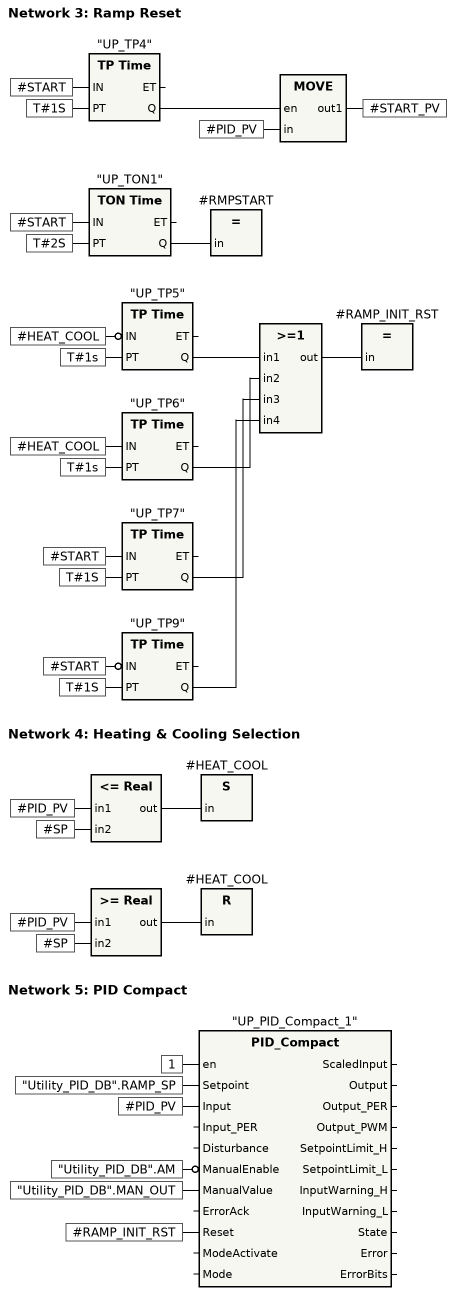
   "UP_TP4".TP(IN := #START, PT := T#1S);
   IF "UP_TP4".Q THEN #START_PV := #PID_PV; END_IF;
   "UP_TON1".TON(IN := #START, PT := T#2S);
   #RMPSTART := "UP_TON1".Q;
   "UP_TP5".TP(IN := NOT #HEAT_COOL, PT := T#1s);
   "UP_TP6".TP(IN := #HEAT_COOL, PT := T#1s);
   "UP_TP7".TP(IN := #START, PT := T#1S);
   "UP_TP9".TP(IN := NOT #START, PT := T#1S);
   #RAMP_INIT_RST := "UP_TP5".Q OR "UP_TP6".Q OR "UP_TP7".Q OR "UP_TP9".Q;
END_REGION

REGION Network 4: Heating & Cooling Selection
   // Heating & Cooling Selection
   IF #PID_PV <= #SP THEN #HEAT_COOL := TRUE; END_IF;
   IF #PID_PV >= #SP THEN #HEAT_COOL := FALSE; END_IF;
END_REGION

REGION Network 5: PID Compact
   IF 1 THEN
       "UP_PID_Compact_1"(Setpoint := "Utility_PID_DB".RAMP_SP,   // PID_Compact
                          Input := #PID_PV,
                          ManualEnable := NOT "Utility_PID_DB".AM,
                          ManualValue := "Utility_PID_DB".MAN_OUT,
                          Reset := #RAMP_INIT_RST);
   END_IF;
END_REGION

REGION Network 6 (SCL): Moving
   (* PID Parameters Moving *)
   "UP_PID_Compact_1".Retain.CtrlParams.Gain:= #P;
   "UP_PID_Compact_1".Retain.CtrlParams.Ti := #I;
   "UP_PID_Compact_1".Retain.CtrlParams.Td := #D;

   #RAMP := #SP;

   IF #RAMP_MODE OR #MASS_CONTROL THEN
       #PID_PV := #PV;
   END_IF;
   IF #JKT_RAMP THEN
       #PID_PV := #JAC_IN;
   END_IF;


   IF #AM = 1 AND #START = 1 AND #SOURCE_SEL<>5 THEN
       #SCVOUT := "UP_PID_Compact_1".Output;
       #CVOUT := "UP_PID_Compact_1".Output_PER;
   END_IF;
   IF (#AM = 1 AND #START = 0 ) OR (#AM = 1 AND #SOURCE_SEL=5) OR (#AM = 1 AND #START=1 AND (#AIR_XV_OPN OR #VENT_OPN OR #DRAIN_XV_OPN)) THEN
       #SCVOUT := 0.0;
       #CVOUT := 0;
   END_IF;
   IF #AM = 0 THEN
       #SCVOUT := "UP_PID_Compact_1".Output;
       #CVOUT := "UP_PID_Compact_1".Output_PER;
   END_IF;

   IF #AM = 1 AND #START = 1 AND #DRAIN_XV_OPN AND #SCV_XV_OPN THEN
       #iSTEAM_SCVOUT := 100.0;
       #iDRAIN_UP := 1;
   ELSE
       #iDRAIN_UP := 0;
   END_IF;
   IF #AM = 1 AND #START = 1 AND #SOURCE_SEL = 5 AND #iDRAIN_UP= 0 THEN
       #iSTEAM_SCVOUT := "UP_PID_Compact_1".Output;
       #iSTEAM_CVOUT := "UP_PID_Compact_1".Output_PER;
   END_IF;
   IF (#AM = 1 AND #START = 0) OR (#AM = 1 AND #SOURCE_SEL <> 5) OR (#AM = 1 AND #START = 1 AND ((#CONDENSATE_XV_OPN AND #SOURCE_SEL <> 5) OR (#AIR_XV_OPN AND #SOURCE_SEL = 5))) THEN
       #iSTEAM_SCVOUT := 0.0;
       #iSTEAM_CVOUT := 0;
   END_IF;


   (* Cooling *)
   IF #HEAT_COOL = 0 AND #START = 1 AND (#RAMP_MODE OR #JKT_RAMP) THEN
       "UP_RampFunction_DB1".PositiveFallingSlewRate := ABS((#START_PV - #SP) / (#TIME*60)); 
       "UP_PID_Compact_1".Config.InvertControl := 1;
   END_IF;
   IF #HEAT_COOL = 0 AND #START = 1 AND #MASS_CONTROL THEN
       "UP_RampFunction_DB1".PositiveFallingSlewRate := ABS((#START_PV - #SP) / (1 * 60));
       "UP_PID_Compact_1".Config.InvertControl := 1;
   END_IF;

   (* Heating *)
   IF #HEAT_COOL = 1 AND #START = 1 AND (#RAMP_MODE OR #JKT_RAMP) THEN
       "UP_RampFunction_DB1".PositiveRisingSlewRate := ABS((#SP - #START_PV) / (#TIME*60)); 
       "UP_PID_Compact_1".Config.InvertControl := 0;
   END_IF;
   IF #HEAT_COOL = 1 AND #START = 1 AND #MASS_CONTROL THEN
       "UP_RampFunction_DB1".PositiveRisingSlewRate := ABS((#SP - #START_PV) / (1 * 60));
       "UP_PID_Compact_1".Config.InvertControl := 0;
   END_IF;
END_REGION

REGION Network 7: OPERATION RUNTIME
   // OPERATION RUNTIME
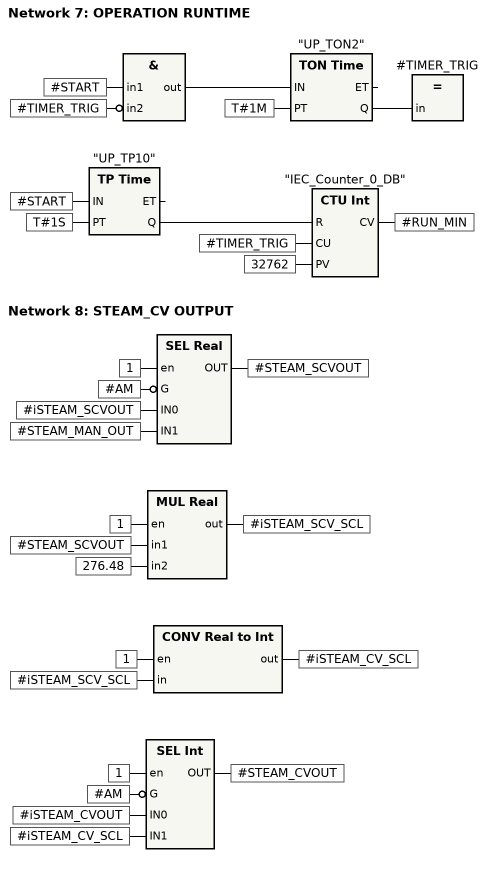
   "UP_TON2".TON(IN := #START AND NOT #TIMER_TRIG, PT := T#1M);
   #TIMER_TRIG := "UP_TON2".Q;
   "UP_TP10".TP(IN := #START, PT := T#1S);
   "IEC_Counter_0_DB".CTU(R := "UP_TP10".Q, CU := #TIMER_TRIG, PV := 32762, CV => #RUN_MIN);
END_REGION

REGION Network 8: STEAM_CV OUTPUT
   IF 1 THEN
       #STEAM_SCVOUT := SEL(G := NOT #AM, IN0 := #iSTEAM_SCVOUT, IN1 := #STEAM_MAN_OUT);
       #iSTEAM_SCV_SCL := #STEAM_SCVOUT * 276.48;
       #iSTEAM_CV_SCL := REAL_TO_INT(#iSTEAM_SCV_SCL);
       #STEAM_CVOUT := SEL(G := NOT #AM, IN0 := #iSTEAM_CVOUT, IN1 := #iSTEAM_CV_SCL);
   END_IF;
END_REGION
END_FUNCTION_BLOCK

FUNCTION_BLOCK "3WayValve"   // FB14, LAD
{ S7_Optimized_Access := 'TRUE' }
VERSION : 0.1
// stored: AutoNumber true, IsIECCheckEnabled false, IsRetainMemResEnabled false, MemoryReserve 100, SetENOAutomatically false, UDAEnableTagReadback false
   VAR_INPUT
      "auto/manual" : Bool;
      v1_open_auto : Bool;
      v1_open_man : Bool;
      v1_fbk_open : Bool;
      v1_fbk_close : Bool;
      v2_open_auto : Bool;
      v2_open_man : Bool;
      v2_fbk_open : Bool;
      reset : Bool;
      intl : Bool;
      monito_time : Time;
      Mon_En : Bool;
   END_VAR
   VAR_OUTPUT
      v1_cmd1 : Bool;
      v2_cmd2 : Bool;
      fault : Bool;
      status : Int;
   END_VAR
   VAR
      open_fault : Bool;
      close_fault : Bool;
      IEC_Timer_0_Instance : TON_TIME;
      IEC_Timer_0_Instance_1 { S7_SetPoint := 'True'} : TON_TIME;
      IEC_Timer_0_Instance_2 { S7_SetPoint := 'True'} : TON_TIME;
      V1_ON : Bool;
   END_VAR
   VAR_TEMP   // added for the SCL form of the ladder/FBD networks
      _w1 : Bool;
   END_VAR
BEGIN

REGION Network 1
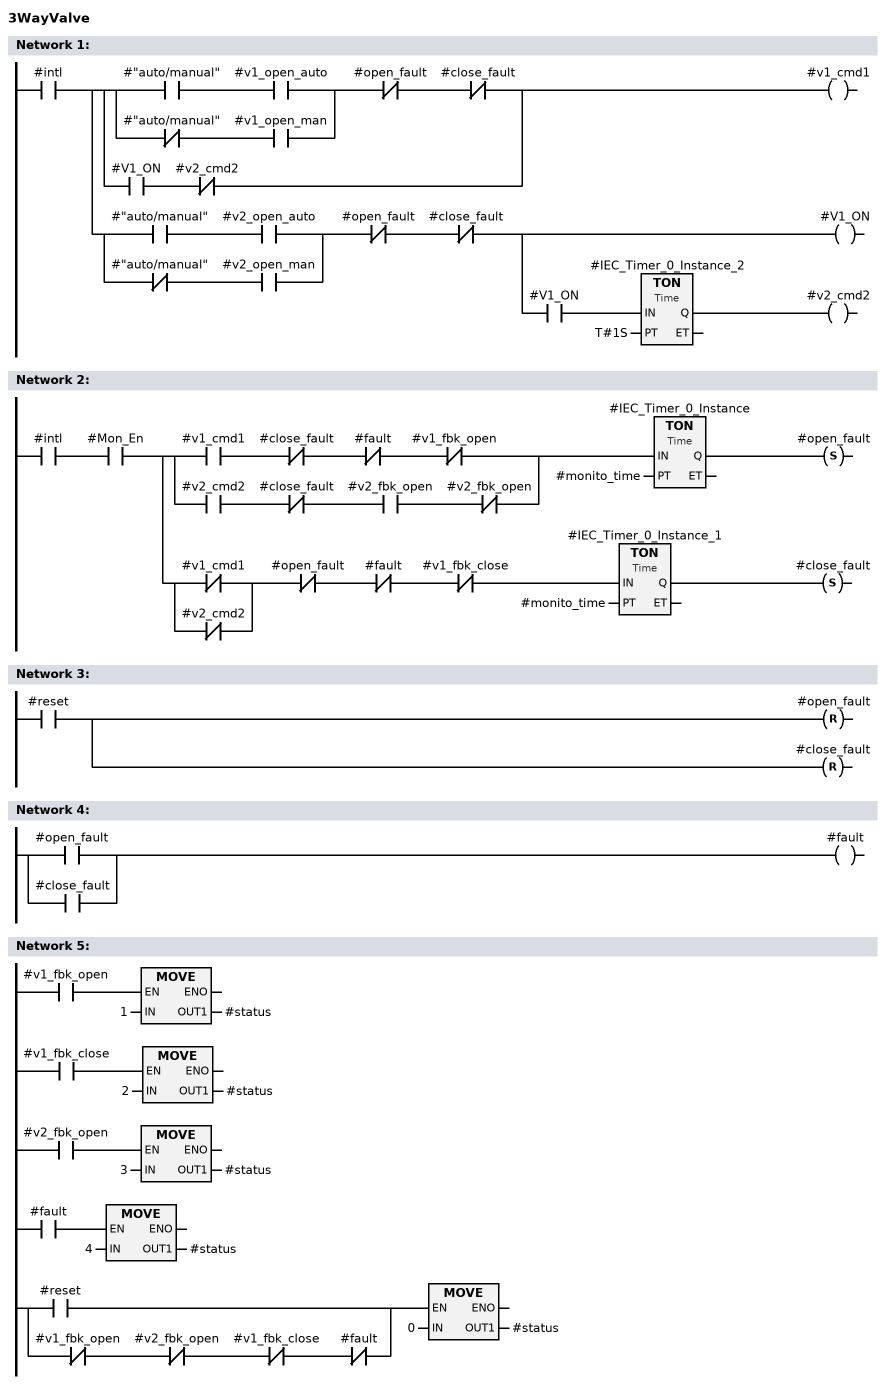
   RUNG wire#powerrail
      Contact( #intl )
      wire#w1
      Contact( #"auto/manual" )
      Contact( #v1_open_auto )
      wire#w2
      I_Contact( #open_fault )
      I_Contact( #close_fault )
      wire#w3
      Coil( #v1_cmd1 )
   END_RUNG
   RUNG wire#w1
      I_Contact( #"auto/manual" )
      Contact( #v1_open_man )
   END_RUNG wire#w2
   RUNG wire#w1
      Contact( #V1_ON )
      I_Contact( #v2_cmd2 )
   END_RUNG wire#w3
   RUNG wire#w1
      Contact( #"auto/manual" )
      Contact( #v2_open_auto )
      wire#w4
      I_Contact( #open_fault )
      I_Contact( #close_fault )
      wire#w5
      Coil( #V1_ON )
   END_RUNG
   RUNG wire#w1
      I_Contact( #"auto/manual" )
      Contact( #v2_open_man )
   END_RUNG wire#w4
   RUNG wire#w5
      Contact( #V1_ON )
      { S7_Templates := "time_type := Time" } #IEC_Timer_0_Instance_2.TON(pt := T#1S, et =>)
      Coil( #v2_cmd2 )
   END_RUNG
   // the same network as SCL:
   #v1_cmd1 := #intl AND ((((#"auto/manual" AND #v1_open_auto) OR (NOT #"auto/manual" AND #v1_open_man)) AND NOT #open_fault AND NOT #close_fault) OR (#V1_ON AND NOT #v2_cmd2));
   #V1_ON := #intl AND ((#"auto/manual" AND #v2_open_auto) OR (NOT #"auto/manual" AND #v2_open_man)) AND NOT #open_fault AND NOT #close_fault;
   #IEC_Timer_0_Instance_2(IN := #V1_ON AND #V1_ON, PT := T#1S);   // TON
   #v2_cmd2 := #IEC_Timer_0_Instance_2.Q;
END_REGION

REGION Network 2
   RUNG wire#powerrail
      Contact( #intl )
      Contact( #Mon_En )
      wire#w1
      Contact( #v1_cmd1 )
      I_Contact( #close_fault )
      I_Contact( #fault )
      I_Contact( #v1_fbk_open )
      wire#w2
      { S7_Templates := "time_type := Time" } #IEC_Timer_0_Instance.TON(pt := #monito_time, et =>)
      S_Coil( #open_fault )
   END_RUNG
   RUNG wire#w1
      Contact( #v2_cmd2 )
      I_Contact( #close_fault )
      Contact( #v2_fbk_open )
      I_Contact( #v2_fbk_open )
   END_RUNG wire#w2
   RUNG wire#w1
      I_Contact( #v1_cmd1 )
      wire#w3
      I_Contact( #open_fault )
      I_Contact( #fault )
      I_Contact( #v1_fbk_close )
      { S7_Templates := "time_type := Time" } #IEC_Timer_0_Instance_1.TON(pt := #monito_time, et =>)
      S_Coil( #close_fault )
   END_RUNG
   RUNG wire#w1
      I_Contact( #v2_cmd2 )
   END_RUNG wire#w3
   // the same network as SCL:
   #_w1 := #intl AND #Mon_En;
   #IEC_Timer_0_Instance(IN := #_w1 AND ((#v1_cmd1 AND NOT #close_fault AND NOT #fault AND NOT #v1_fbk_open) OR (#v2_cmd2 AND NOT #close_fault AND #v2_fbk_open AND NOT #v2_fbk_open)),   // TON
                         PT := #monito_time);
   IF #IEC_Timer_0_Instance.Q THEN #open_fault := TRUE; END_IF;
   #IEC_Timer_0_Instance_1(IN := #_w1 AND (NOT #v1_cmd1 OR NOT #v2_cmd2) AND NOT #open_fault AND NOT #fault AND NOT #v1_fbk_close,   // TON
                           PT := #monito_time);
   IF #IEC_Timer_0_Instance_1.Q THEN #close_fault := TRUE; END_IF;
END_REGION

REGION Network 3
   RUNG wire#powerrail
      Contact( #reset )
      wire#w1
      R_Coil( #open_fault )
   END_RUNG
   RUNG wire#w1
      R_Coil( #close_fault )
   END_RUNG
   // the same network as SCL:
   IF #reset THEN
       #open_fault := FALSE;
       #close_fault := FALSE;
   END_IF;
END_REGION

REGION Network 4
   RUNG wire#powerrail
      Contact( #open_fault )
      wire#w1
      Coil( #fault )
   END_RUNG
   RUNG wire#powerrail
      Contact( #close_fault )
   END_RUNG wire#w1
   // the same network as SCL:
   #fault := #open_fault OR #close_fault;
END_REGION

REGION Network 5
   RUNG wire#powerrail
      Contact( #v1_fbk_open )
      Move(in := 1, out1 => #status)
   END_RUNG
   RUNG wire#powerrail
      Contact( #v1_fbk_close )
      Move(in := 2, out1 => #status)
   END_RUNG
   RUNG wire#powerrail
      Contact( #v2_fbk_open )
      Move(in := 3, out1 => #status)
   END_RUNG
   RUNG wire#powerrail
      Contact( #fault )
      Move(in := 4, out1 => #status)
   END_RUNG
   RUNG wire#powerrail
      Contact( #reset )
      wire#w1
      Move(in := 0, out1 => #status)
   END_RUNG
   RUNG wire#powerrail
      I_Contact( #v1_fbk_open )
      I_Contact( #v2_fbk_open )
      I_Contact( #v1_fbk_close )
      I_Contact( #fault )
   END_RUNG wire#w1
   // the same network as SCL:
   IF #v1_fbk_open THEN #status := 1; END_IF;
   IF #v1_fbk_close THEN #status := 2; END_IF;
   IF #v2_fbk_open THEN #status := 3; END_IF;
   IF #fault THEN #status := 4; END_IF;
   IF #reset OR (NOT #v1_fbk_open AND NOT #v2_fbk_open AND NOT #v1_fbk_close AND NOT #fault) THEN
       #status := 0;
   END_IF;
END_REGION
END_FUNCTION_BLOCK

DATA_BLOCK "Utility_PID_DB"   // DB3
VERSION : 0.1
// stored: AutoNumber true, DBAccessibleFromOPCUA true, DBAccessibleFromWebserver true, InstanceOfName Utility_PID, InstanceOfType FB
"Utility_PID"
BEGIN
END_DATA_BLOCK

DATA_BLOCK "Utility_PID_DB_1"   // DB197
VERSION : 0.1
// stored: AutoNumber true, DBAccessibleFromOPCUA true, DBAccessibleFromWebserver true, InstanceOfName Utility_PID, InstanceOfType FB
"Utility_PID"
BEGIN
END_DATA_BLOCK

DATA_BLOCK "Utility_PID_DB_2"   // DB198
VERSION : 0.1
// stored: AutoNumber true, DBAccessibleFromOPCUA true, DBAccessibleFromWebserver true, InstanceOfName Utility_PID, InstanceOfType FB
"Utility_PID"
BEGIN
END_DATA_BLOCK

DATA_BLOCK "Utility_PID_DB_3"   // DB199
VERSION : 0.1
// stored: AutoNumber true, DBAccessibleFromOPCUA true, DBAccessibleFromWebserver true, InstanceOfName Utility_PID, InstanceOfType FB
"Utility_PID"
BEGIN
END_DATA_BLOCK

DATA_BLOCK "Utility_selection_DB"   // DB6
VERSION : 0.1
// stored: AutoNumber true, DBAccessibleFromOPCUA true, DBAccessibleFromWebserver true, InstanceOfName Utility_selection, InstanceOfType FB
"Utility_selection"
BEGIN
END_DATA_BLOCK

DATA_BLOCK "3WayValve_DB"   // DB108
VERSION : 0.1
// stored: AutoNumber true, DBAccessibleFromOPCUA true, DBAccessibleFromWebserver true, InstanceOfName 3WayValve, InstanceOfType FB
"3WayValve"
BEGIN
END_DATA_BLOCK

DATA_BLOCK "valve_DB"   // DB116
VERSION : 0.1
// stored: AutoNumber true, DBAccessibleFromOPCUA true, DBAccessibleFromWebserver true, InstanceOfName valve, InstanceOfType FB
"valve"
BEGIN
END_DATA_BLOCK

DATA_BLOCK "HOOTER_DB"   // DB115
VERSION : 0.1
// stored: AutoNumber true, DBAccessibleFromOPCUA true, DBAccessibleFromWebserver true, InstanceOfName HOOTER, InstanceOfType FB
"HOOTER"
BEGIN
END_DATA_BLOCK

DATA_BLOCK "HOOTER_DB_1"   // DB102
VERSION : 0.1
// stored: AutoNumber true, DBAccessibleFromOPCUA true, DBAccessibleFromWebserver true, InstanceOfName HOOTER, InstanceOfType FB
"HOOTER"
BEGIN
END_DATA_BLOCK

DATA_BLOCK "HOOTER_RT1"   // DB104
// stored: AutoNumber true, DBAccessibleFromOPCUA true, DBAccessibleFromWebserver true, InstanceOfName R_TRIG, OfSystemLibElement R_TRIG, OfSystemLibVersion 1.0
"R_TRIG"
   // VAR_INPUT
   //    CLK : Bool;
   // END_VAR
   // VAR_OUTPUT
   //    Q : Bool;
   // END_VAR
   // VAR
   //    Stat_Bit : Bool;
   // END_VAR
BEGIN
END_DATA_BLOCK

DATA_BLOCK "HOOTER_RT10"   // DB114
// stored: AutoNumber true, DBAccessibleFromOPCUA true, DBAccessibleFromWebserver true, InstanceOfName R_TRIG, OfSystemLibElement R_TRIG, OfSystemLibVersion 1.0
"R_TRIG"
   // VAR_INPUT
   //    CLK : Bool;
   // END_VAR
   // VAR_OUTPUT
   //    Q : Bool;
   // END_VAR
   // VAR
   //    Stat_Bit : Bool;
   // END_VAR
BEGIN
END_DATA_BLOCK

DATA_BLOCK "HOOTER_RT2"   // DB105
// stored: AutoNumber true, DBAccessibleFromOPCUA true, DBAccessibleFromWebserver true, InstanceOfName R_TRIG, OfSystemLibElement R_TRIG, OfSystemLibVersion 1.0
"R_TRIG"
   // VAR_INPUT
   //    CLK : Bool;
   // END_VAR
   // VAR_OUTPUT
   //    Q : Bool;
   // END_VAR
   // VAR
   //    Stat_Bit : Bool;
   // END_VAR
BEGIN
END_DATA_BLOCK

DATA_BLOCK "HOOTER_RT3"   // DB106
// stored: AutoNumber true, DBAccessibleFromOPCUA true, DBAccessibleFromWebserver true, InstanceOfName R_TRIG, OfSystemLibElement R_TRIG, OfSystemLibVersion 1.0
"R_TRIG"
   // VAR_INPUT
   //    CLK : Bool;
   // END_VAR
   // VAR_OUTPUT
   //    Q : Bool;
   // END_VAR
   // VAR
   //    Stat_Bit : Bool;
   // END_VAR
BEGIN
END_DATA_BLOCK

DATA_BLOCK "HOOTER_RT4"   // DB107
// stored: AutoNumber true, DBAccessibleFromOPCUA true, DBAccessibleFromWebserver true, InstanceOfName R_TRIG, OfSystemLibElement R_TRIG, OfSystemLibVersion 1.0
"R_TRIG"
   // VAR_INPUT
   //    CLK : Bool;
   // END_VAR
   // VAR_OUTPUT
   //    Q : Bool;
   // END_VAR
   // VAR
   //    Stat_Bit : Bool;
   // END_VAR
BEGIN
END_DATA_BLOCK

DATA_BLOCK "HOOTER_RT5"   // DB109
// stored: AutoNumber true, DBAccessibleFromOPCUA true, DBAccessibleFromWebserver true, InstanceOfName R_TRIG, OfSystemLibElement R_TRIG, OfSystemLibVersion 1.0
"R_TRIG"
   // VAR_INPUT
   //    CLK : Bool;
   // END_VAR
   // VAR_OUTPUT
   //    Q : Bool;
   // END_VAR
   // VAR
   //    Stat_Bit : Bool;
   // END_VAR
BEGIN
END_DATA_BLOCK

DATA_BLOCK "HOOTER_RT6"   // DB110
// stored: AutoNumber true, DBAccessibleFromOPCUA true, DBAccessibleFromWebserver true, InstanceOfName R_TRIG, OfSystemLibElement R_TRIG, OfSystemLibVersion 1.0
"R_TRIG"
   // VAR_INPUT
   //    CLK : Bool;
   // END_VAR
   // VAR_OUTPUT
   //    Q : Bool;
   // END_VAR
   // VAR
   //    Stat_Bit : Bool;
   // END_VAR
BEGIN
END_DATA_BLOCK

DATA_BLOCK "HOOTER_RT7"   // DB111
// stored: AutoNumber true, DBAccessibleFromOPCUA true, DBAccessibleFromWebserver true, InstanceOfName R_TRIG, OfSystemLibElement R_TRIG, OfSystemLibVersion 1.0
"R_TRIG"
   // VAR_INPUT
   //    CLK : Bool;
   // END_VAR
   // VAR_OUTPUT
   //    Q : Bool;
   // END_VAR
   // VAR
   //    Stat_Bit : Bool;
   // END_VAR
BEGIN
END_DATA_BLOCK

DATA_BLOCK "HOOTER_RT8"   // DB112
// stored: AutoNumber true, DBAccessibleFromOPCUA true, DBAccessibleFromWebserver true, InstanceOfName R_TRIG, OfSystemLibElement R_TRIG, OfSystemLibVersion 1.0
"R_TRIG"
   // VAR_INPUT
   //    CLK : Bool;
   // END_VAR
   // VAR_OUTPUT
   //    Q : Bool;
   // END_VAR
   // VAR
   //    Stat_Bit : Bool;
   // END_VAR
BEGIN
END_DATA_BLOCK

DATA_BLOCK "HOOTER_RT9"   // DB113
// stored: AutoNumber true, DBAccessibleFromOPCUA true, DBAccessibleFromWebserver true, InstanceOfName R_TRIG, OfSystemLibElement R_TRIG, OfSystemLibVersion 1.0
"R_TRIG"
   // VAR_INPUT
   //    CLK : Bool;
   // END_VAR
   // VAR_OUTPUT
   //    Q : Bool;
   // END_VAR
   // VAR
   //    Stat_Bit : Bool;
   // END_VAR
BEGIN
END_DATA_BLOCK

DATA_BLOCK "IEC_Counter_0_DB"   // DB18
{ S7_Optimized_Access := 'TRUE' }
// stored: AutoNumber true, DBAccessibleFromOPCUA true, DBAccessibleFromWebserver true, InstanceOfName IEC_COUNTER, OfSystemLibElement IEC_COUNTER, OfSystemLibVersion 1.0
"IEC_COUNTER"
   // VAR RETAIN
   //    CU : Bool;
   //    CD : Bool;
   //    R : Bool;
   //    LD : Bool;
   //    QU : Bool;
   //    QD : Bool;
   //    PV : Int;
   //    CV : Int;
   // END_VAR
BEGIN
END_DATA_BLOCK

DATA_BLOCK "Precheck_TP1"   // DB84
{ S7_Optimized_Access := 'TRUE' }
// stored: AutoNumber true, DBAccessibleFromOPCUA true, DBAccessibleFromWebserver true, InstanceOfName IEC_TIMER, OfSystemLibElement IEC_TIMER, OfSystemLibVersion 1.0
"IEC_TIMER"
   // VAR
   //    PT : Time;
   //    ET { ExternalWritable := 'False'} : Time;
   //    IN : Bool;
   //    Q { ExternalWritable := 'False'} : Bool;
   // END_VAR
BEGIN
END_DATA_BLOCK

DATA_BLOCK "Precheck_TP2"   // DB85
{ S7_Optimized_Access := 'TRUE' }
// stored: AutoNumber true, DBAccessibleFromOPCUA true, DBAccessibleFromWebserver true, InstanceOfName IEC_TIMER, OfSystemLibElement IEC_TIMER, OfSystemLibVersion 1.0
"IEC_TIMER"
   // VAR
   //    PT : Time;
   //    ET { ExternalWritable := 'False'} : Time;
   //    IN : Bool;
   //    Q { ExternalWritable := 'False'} : Bool;
   // END_VAR
BEGIN
END_DATA_BLOCK

DATA_BLOCK "Precheck_TP3"   // DB86
{ S7_Optimized_Access := 'TRUE' }
// stored: AutoNumber true, DBAccessibleFromOPCUA true, DBAccessibleFromWebserver true, InstanceOfName IEC_TIMER, OfSystemLibElement IEC_TIMER, OfSystemLibVersion 1.0
"IEC_TIMER"
   // VAR
   //    PT : Time;
   //    ET { ExternalWritable := 'False'} : Time;
   //    IN : Bool;
   //    Q { ExternalWritable := 'False'} : Bool;
   // END_VAR
BEGIN
END_DATA_BLOCK

DATA_BLOCK "Precheck_TP4"   // DB87
{ S7_Optimized_Access := 'TRUE' }
// stored: AutoNumber true, DBAccessibleFromOPCUA true, DBAccessibleFromWebserver true, InstanceOfName IEC_TIMER, OfSystemLibElement IEC_TIMER, OfSystemLibVersion 1.0
"IEC_TIMER"
   // VAR
   //    PT : Time;
   //    ET { ExternalWritable := 'False'} : Time;
   //    IN : Bool;
   //    Q { ExternalWritable := 'False'} : Bool;
   // END_VAR
BEGIN
END_DATA_BLOCK

DATA_BLOCK "Precheck_TP5"   // DB88
{ S7_Optimized_Access := 'TRUE' }
// stored: AutoNumber true, DBAccessibleFromOPCUA true, DBAccessibleFromWebserver true, InstanceOfName IEC_TIMER, OfSystemLibElement IEC_TIMER, OfSystemLibVersion 1.0
"IEC_TIMER"
   // VAR
   //    PT : Time;
   //    ET { ExternalWritable := 'False'} : Time;
   //    IN : Bool;
   //    Q { ExternalWritable := 'False'} : Bool;
   // END_VAR
BEGIN
END_DATA_BLOCK

DATA_BLOCK "Precheck_TP6"   // DB89
{ S7_Optimized_Access := 'TRUE' }
// stored: AutoNumber true, DBAccessibleFromOPCUA true, DBAccessibleFromWebserver true, InstanceOfName IEC_TIMER, OfSystemLibElement IEC_TIMER, OfSystemLibVersion 1.0
"IEC_TIMER"
   // VAR
   //    PT : Time;
   //    ET { ExternalWritable := 'False'} : Time;
   //    IN : Bool;
   //    Q { ExternalWritable := 'False'} : Bool;
   // END_VAR
BEGIN
END_DATA_BLOCK

DATA_BLOCK "Precheck_TP7"   // DB103
{ S7_Optimized_Access := 'TRUE' }
// stored: AutoNumber true, DBAccessibleFromOPCUA true, DBAccessibleFromWebserver true, InstanceOfName IEC_TIMER, OfSystemLibElement IEC_TIMER, OfSystemLibVersion 1.0
"IEC_TIMER"
   // VAR
   //    PT : Time;
   //    ET { ExternalWritable := 'False'} : Time;
   //    IN : Bool;
   //    Q { ExternalWritable := 'False'} : Bool;
   // END_VAR
BEGIN
END_DATA_BLOCK

DATA_BLOCK "RESET_TP1"   // DB100
{ S7_Optimized_Access := 'TRUE' }
// stored: AutoNumber true, DBAccessibleFromOPCUA true, DBAccessibleFromWebserver true, InstanceOfName IEC_TIMER, OfSystemLibElement IEC_TIMER, OfSystemLibVersion 1.0
"IEC_TIMER"
   // VAR
   //    PT : Time;
   //    ET { ExternalWritable := 'False'} : Time;
   //    IN : Bool;
   //    Q { ExternalWritable := 'False'} : Bool;
   // END_VAR
BEGIN
END_DATA_BLOCK

DATA_BLOCK "SS_FT1"   // DB56
// stored: AutoNumber true, DBAccessibleFromOPCUA true, DBAccessibleFromWebserver true, InstanceOfName F_TRIG, OfSystemLibElement F_TRIG, OfSystemLibVersion 1.0
"F_TRIG"
   // VAR_INPUT
   //    CLK : Bool;
   // END_VAR
   // VAR_OUTPUT
   //    Q : Bool;
   // END_VAR
   // VAR
   //    Stat_Bit : Bool;
   // END_VAR
BEGIN
END_DATA_BLOCK

DATA_BLOCK "SS_TON2"   // DB61
{ S7_Optimized_Access := 'TRUE' }
// stored: AutoNumber true, DBAccessibleFromOPCUA true, DBAccessibleFromWebserver true, InstanceOfName IEC_TIMER, OfSystemLibElement IEC_TIMER, OfSystemLibVersion 1.0
"IEC_TIMER"
   // VAR
   //    PT : Time;
   //    ET { ExternalWritable := 'False'} : Time;
   //    IN : Bool;
   //    Q { ExternalWritable := 'False'} : Bool;
   // END_VAR
BEGIN
END_DATA_BLOCK

DATA_BLOCK "UP_TON1"   // DB11
{ S7_Optimized_Access := 'TRUE' }
// stored: AutoNumber true, DBAccessibleFromOPCUA true, DBAccessibleFromWebserver true, InstanceOfName IEC_TIMER, OfSystemLibElement IEC_TIMER, OfSystemLibVersion 1.0
"IEC_TIMER"
   // VAR
   //    PT : Time;
   //    ET { ExternalWritable := 'False'} : Time;
   //    IN : Bool;
   //    Q { ExternalWritable := 'False'} : Bool;
   // END_VAR
BEGIN
END_DATA_BLOCK

DATA_BLOCK "UP_TON2"   // DB20
{ S7_Optimized_Access := 'TRUE' }
// stored: AutoNumber true, DBAccessibleFromOPCUA true, DBAccessibleFromWebserver true, InstanceOfName IEC_TIMER, OfSystemLibElement IEC_TIMER, OfSystemLibVersion 1.0
"IEC_TIMER"
   // VAR
   //    PT : Time;
   //    ET { ExternalWritable := 'False'} : Time;
   //    IN : Bool;
   //    Q { ExternalWritable := 'False'} : Bool;
   // END_VAR
BEGIN
END_DATA_BLOCK

DATA_BLOCK "UP_TP1"   // DB2
{ S7_Optimized_Access := 'TRUE' }
// stored: AutoNumber true, DBAccessibleFromOPCUA true, DBAccessibleFromWebserver true, InstanceOfName IEC_TIMER, OfSystemLibElement IEC_TIMER, OfSystemLibVersion 1.0
"IEC_TIMER"
   // VAR
   //    PT : Time;
   //    ET { ExternalWritable := 'False'} : Time;
   //    IN : Bool;
   //    Q { ExternalWritable := 'False'} : Bool;
   // END_VAR
BEGIN
END_DATA_BLOCK

DATA_BLOCK "UP_TP10"   // DB21
{ S7_Optimized_Access := 'TRUE' }
// stored: AutoNumber true, DBAccessibleFromOPCUA true, DBAccessibleFromWebserver true, InstanceOfName IEC_TIMER, OfSystemLibElement IEC_TIMER, OfSystemLibVersion 1.0
"IEC_TIMER"
   // VAR
   //    PT : Time;
   //    ET { ExternalWritable := 'False'} : Time;
   //    IN : Bool;
   //    Q { ExternalWritable := 'False'} : Bool;
   // END_VAR
BEGIN
END_DATA_BLOCK

DATA_BLOCK "UP_TP2"   // DB4
{ S7_Optimized_Access := 'TRUE' }
// stored: AutoNumber true, DBAccessibleFromOPCUA true, DBAccessibleFromWebserver true, InstanceOfName IEC_TIMER, OfSystemLibElement IEC_TIMER, OfSystemLibVersion 1.0
"IEC_TIMER"
   // VAR
   //    PT : Time;
   //    ET { ExternalWritable := 'False'} : Time;
   //    IN : Bool;
   //    Q { ExternalWritable := 'False'} : Bool;
   // END_VAR
BEGIN
END_DATA_BLOCK

DATA_BLOCK "UP_TP4"   // DB10
{ S7_Optimized_Access := 'TRUE' }
// stored: AutoNumber true, DBAccessibleFromOPCUA true, DBAccessibleFromWebserver true, InstanceOfName IEC_TIMER, OfSystemLibElement IEC_TIMER, OfSystemLibVersion 1.0
"IEC_TIMER"
   // VAR
   //    PT : Time;
   //    ET { ExternalWritable := 'False'} : Time;
   //    IN : Bool;
   //    Q { ExternalWritable := 'False'} : Bool;
   // END_VAR
BEGIN
END_DATA_BLOCK

DATA_BLOCK "UP_TP5"   // DB12
{ S7_Optimized_Access := 'TRUE' }
// stored: AutoNumber true, DBAccessibleFromOPCUA true, DBAccessibleFromWebserver true, InstanceOfName IEC_TIMER, OfSystemLibElement IEC_TIMER, OfSystemLibVersion 1.0
"IEC_TIMER"
   // VAR
   //    PT : Time;
   //    ET { ExternalWritable := 'False'} : Time;
   //    IN : Bool;
   //    Q { ExternalWritable := 'False'} : Bool;
   // END_VAR
BEGIN
END_DATA_BLOCK

DATA_BLOCK "UP_TP6"   // DB13
{ S7_Optimized_Access := 'TRUE' }
// stored: AutoNumber true, DBAccessibleFromOPCUA true, DBAccessibleFromWebserver true, InstanceOfName IEC_TIMER, OfSystemLibElement IEC_TIMER, OfSystemLibVersion 1.0
"IEC_TIMER"
   // VAR
   //    PT : Time;
   //    ET { ExternalWritable := 'False'} : Time;
   //    IN : Bool;
   //    Q { ExternalWritable := 'False'} : Bool;
   // END_VAR
BEGIN
END_DATA_BLOCK

DATA_BLOCK "UP_TP7"   // DB14
{ S7_Optimized_Access := 'TRUE' }
// stored: AutoNumber true, DBAccessibleFromOPCUA true, DBAccessibleFromWebserver true, InstanceOfName IEC_TIMER, OfSystemLibElement IEC_TIMER, OfSystemLibVersion 1.0
"IEC_TIMER"
   // VAR
   //    PT : Time;
   //    ET { ExternalWritable := 'False'} : Time;
   //    IN : Bool;
   //    Q { ExternalWritable := 'False'} : Bool;
   // END_VAR
BEGIN
END_DATA_BLOCK

DATA_BLOCK "UP_TP8"   // DB16
{ S7_Optimized_Access := 'TRUE' }
// stored: AutoNumber true, DBAccessibleFromOPCUA true, DBAccessibleFromWebserver true, InstanceOfName IEC_TIMER, OfSystemLibElement IEC_TIMER, OfSystemLibVersion 1.0
"IEC_TIMER"
   // VAR
   //    PT : Time;
   //    ET { ExternalWritable := 'False'} : Time;
   //    IN : Bool;
   //    Q { ExternalWritable := 'False'} : Bool;
   // END_VAR
BEGIN
END_DATA_BLOCK

DATA_BLOCK "UP_TP9"   // DB17
{ S7_Optimized_Access := 'TRUE' }
// stored: AutoNumber true, DBAccessibleFromOPCUA true, DBAccessibleFromWebserver true, InstanceOfName IEC_TIMER, OfSystemLibElement IEC_TIMER, OfSystemLibVersion 1.0
"IEC_TIMER"
   // VAR
   //    PT : Time;
   //    ET { ExternalWritable := 'False'} : Time;
   //    IN : Bool;
   //    Q { ExternalWritable := 'False'} : Bool;
   // END_VAR
BEGIN
END_DATA_BLOCK

DATA_BLOCK "US_TON1"   // DB34
{ S7_Optimized_Access := 'TRUE' }
// stored: AutoNumber true, DBAccessibleFromOPCUA true, DBAccessibleFromWebserver true, InstanceOfName IEC_TIMER, OfSystemLibElement IEC_TIMER, OfSystemLibVersion 1.0
"IEC_TIMER"
   // VAR
   //    PT : Time;
   //    ET { ExternalWritable := 'False'} : Time;
   //    IN : Bool;
   //    Q { ExternalWritable := 'False'} : Bool;
   // END_VAR
BEGIN
END_DATA_BLOCK

DATA_BLOCK "HSSR_019_CV103"   // DB83
// stored: AutoNumber true, DBAccessibleFromOPCUA true, DBAccessibleFromWebserver true, InstanceOfName PID_Compact, OfSystemLibElement PID_Compact, OfSystemLibVersion 2.4
PID_Compact   // technology object, version 2.4
   // VAR_INPUT
   //    Setpoint : Real;
   //    Input : Real;
   //    Input_PER : Int;
   //    Disturbance : Real;
   //    ManualEnable : Bool;
   //    ManualValue : Real;
   //    ErrorAck : Bool;
   //    Reset : Bool;
   //    ModeActivate : Bool;
   // END_VAR
   // VAR_OUTPUT
   //    ScaledInput { ExternalWritable := 'False'} : Real;
   //    Output { ExternalWritable := 'False'} : Real;
   //    Output_PER { ExternalWritable := 'False'} : Int;
   //    Output_PWM { ExternalWritable := 'False'} : Bool;
   //    SetpointLimit_H { ExternalWritable := 'False'} : Bool;
   //    SetpointLimit_L { ExternalWritable := 'False'} : Bool;
   //    InputWarning_H { ExternalWritable := 'False'} : Bool;
   //    InputWarning_L { ExternalWritable := 'False'} : Bool;
   //    State { ExternalWritable := 'False'} : Int;
   //    Error { ExternalWritable := 'False'} : Bool;
   //    ErrorBits { ExternalWritable := 'False'} : DWord;
   // END_VAR
   // VAR_IN_OUT
   //    Mode : Int;
   // END_VAR
   // VAR
   //    InternalDiagnostic : DWord;
   //    InternalVersion { ExternalWritable := 'False'} : DWord;
   //    InternalRTVersion : DWord;
   //    IntegralResetMode { S7_SetPoint := 'True'} : Int;
   //    OverwriteInitialOutputValue : Real;
   //    RunModeByStartup { S7_SetPoint := 'True'} : Bool;
   //    LoadBackUp : Bool;
   //    SetSubstituteOutput { S7_SetPoint := 'True'} : Bool;
   //    PhysicalUnit { ExternalWritable := 'False'; S7_SetPoint := 'True'} : Int;
   //    PhysicalQuantity { ExternalWritable := 'False'; S7_SetPoint := 'True'} : Int;
   //    ActivateRecoverMode { S7_SetPoint := 'True'} : Bool;
   // END_VAR
   // VAR RETAIN
   //    Warning { ExternalWritable := 'False'} : DWord;
   //    WarningInternal { ExternalWritable := 'False'} : DWord;
   // END_VAR
   // VAR
   //    Progress { ExternalWritable := 'False'} : Real;
   //    CurrentSetpoint { ExternalWritable := 'False'} : Real;
   //    CancelTuningLevel { S7_SetPoint := 'True'} : Real;
   //    SubstituteOutput { S7_SetPoint := 'True'} : Real;
   //    Config { S7_SetPoint := 'True'} : PID_CompactConfig;
   //    CycleTime { S7_SetPoint := 'True'} : PID_CycleTime;
   //    CtrlParamsBackUp { S7_SetPoint := 'True'} : PID_CompactControlParams;
   //    PIDSelfTune { S7_SetPoint := 'True'} : PID_CompactSelfTune;
   //    PIDCtrl { S7_SetPoint := 'True'} : PID_CompactControl;
   // END_VAR
   // VAR RETAIN
   //    Retain { S7_SetPoint := 'True'} : PID_CompactRetain;
   // END_VAR
BEGIN
END_DATA_BLOCK

DATA_BLOCK "UP_PID_Compact_1"   // DB15
// stored: AutoNumber true, DBAccessibleFromOPCUA true, DBAccessibleFromWebserver true, InstanceOfName PID_Compact, OfSystemLibElement PID_Compact, OfSystemLibVersion 2.4
PID_Compact   // technology object, version 2.4
   // VAR_INPUT
   //    Setpoint : Real;
   //    Input : Real;
   //    Input_PER : Int;
   //    Disturbance : Real;
   //    ManualEnable : Bool;
   //    ManualValue : Real;
   //    ErrorAck : Bool;
   //    Reset : Bool;
   //    ModeActivate : Bool;
   // END_VAR
   // VAR_OUTPUT
   //    ScaledInput { ExternalWritable := 'False'} : Real;
   //    Output { ExternalWritable := 'False'} : Real;
   //    Output_PER { ExternalWritable := 'False'} : Int;
   //    Output_PWM { ExternalWritable := 'False'} : Bool;
   //    SetpointLimit_H { ExternalWritable := 'False'} : Bool;
   //    SetpointLimit_L { ExternalWritable := 'False'} : Bool;
   //    InputWarning_H { ExternalWritable := 'False'} : Bool;
   //    InputWarning_L { ExternalWritable := 'False'} : Bool;
   //    State { ExternalWritable := 'False'} : Int;
   //    Error { ExternalWritable := 'False'} : Bool;
   //    ErrorBits { ExternalWritable := 'False'} : DWord;
   // END_VAR
   // VAR_IN_OUT
   //    Mode : Int := 3;
   // END_VAR
   // VAR
   //    InternalDiagnostic : DWord;
   //    InternalVersion { ExternalWritable := 'False'} : DWord;
   //    InternalRTVersion : DWord;
   //    IntegralResetMode { S7_SetPoint := 'True'} : Int;
   //    OverwriteInitialOutputValue : Real;
   //    RunModeByStartup { S7_SetPoint := 'True'} : Bool;
   //    LoadBackUp : Bool;
   //    SetSubstituteOutput { S7_SetPoint := 'True'} : Bool;
   //    PhysicalUnit { ExternalWritable := 'False'; S7_SetPoint := 'True'} : Int;
   //    PhysicalQuantity { ExternalWritable := 'False'; S7_SetPoint := 'True'} : Int;
   //    ActivateRecoverMode { S7_SetPoint := 'True'} : Bool;
   // END_VAR
   // VAR RETAIN
   //    Warning { ExternalWritable := 'False'} : DWord;
   //    WarningInternal { ExternalWritable := 'False'} : DWord;
   // END_VAR
   // VAR
   //    Progress { ExternalWritable := 'False'} : Real;
   //    CurrentSetpoint { ExternalWritable := 'False'} : Real;
   //    CancelTuningLevel { S7_SetPoint := 'True'} : Real;
   //    SubstituteOutput { S7_SetPoint := 'True'} : Real;
   //    Config { S7_SetPoint := 'True'} : PID_CompactConfig;
   //    CycleTime { S7_SetPoint := 'True'} : PID_CycleTime;
   //    CtrlParamsBackUp { S7_SetPoint := 'True'} : PID_CompactControlParams;
   //    PIDSelfTune { S7_SetPoint := 'True'} : PID_CompactSelfTune;
   //    PIDCtrl { S7_SetPoint := 'True'} : PID_CompactControl;
   // END_VAR
   // VAR RETAIN
   //    Retain { S7_SetPoint := 'True'} : PID_CompactRetain;
   // END_VAR
BEGIN
END_DATA_BLOCK
